PROGRAM MAIN
VAR
		ESTACION: FB_Estacion;
END_VAR

ESTACION();

END_PROGRAM

(* stored: Version 1.1.0.1, ProductVersion 3.1.4024.12
   POU MAIN: Id {cc42d543-bc9f-4b18-8372-30990ef64672}, SpecialFunc None *)
